(* PLC project TON_TEST, Actility iec61131 1.0.26, author Laurent Nicq *)
(* stored: creationDateTime 2013-01-02T13:55:36, version 1.0.0, modificationDateTime 2013-07-30T14:58:25 *)

PROGRAM main
  VAR_EXTERNAL
    SENSOR : BOOL;
    START : BOOL;
  END_VAR
  VAR
    DELAY : TIME := T#10s;
    Counter : TIME;
  END_VAR
  VAR_EXTERNAL
    TimeElapsed : BOOL;
  END_VAR
  VAR
    OnDelay : TON;
  END_VAR

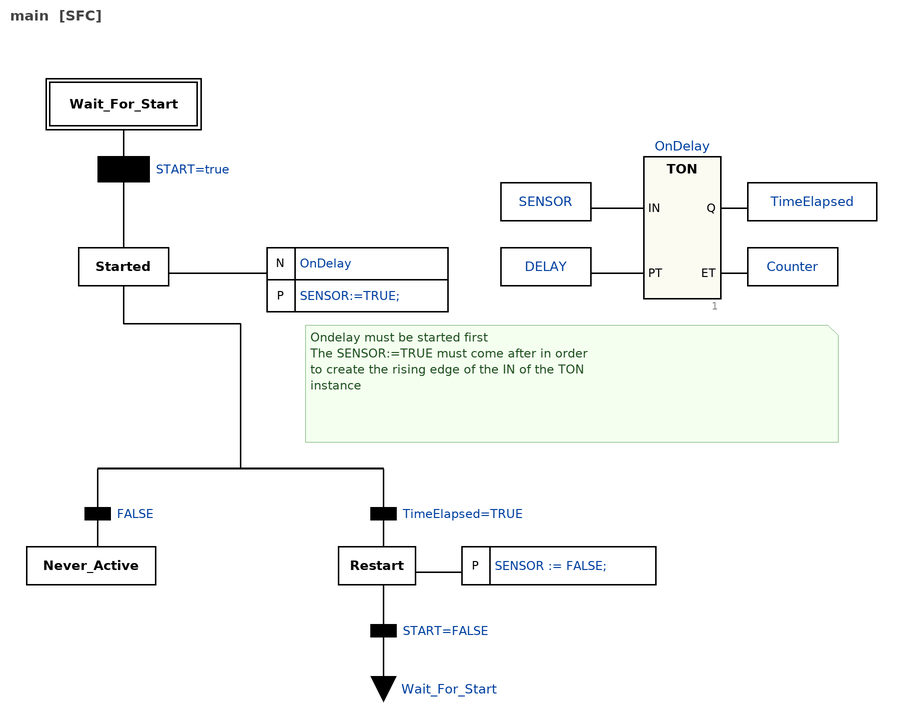
(* Ondelay must be started first
The SENSOR:=TRUE must come after in order
to create the rising edge of the IN of the TON
instance *)
INITIAL_STEP Wait_For_Start:
  COMPUTE_FUNCTION_BLOCKS(S);
END_STEP
TRANSITION FROM Wait_For_Start TO Started
  := START=true;
END_TRANSITION
STEP Started:
  OnDelay(N);
  STARTED_INLINE1(P);
END_STEP
ACTION STARTED_INLINE1:
  SENSOR:=TRUE;
END_ACTION
TRANSITION FROM Started TO Never_Active
  := FALSE;
END_TRANSITION
TRANSITION FROM Started TO Restart
  := TimeElapsed=TRUE;
END_TRANSITION
STEP Never_Active:
END_STEP
STEP Restart:
  RESTART_INLINE2(P);
END_STEP
ACTION RESTART_INLINE2:
  SENSOR := FALSE;
END_ACTION
TRANSITION FROM Restart TO Wait_For_Start
  := START=FALSE;
END_TRANSITION
ACTION COMPUTE_FUNCTION_BLOCKS:  (* blocks drawn on the SFC sheet *)
  OnDelay(IN := SENSOR, PT := DELAY);
  TimeElapsed := OnDelay.Q;
  Counter := OnDelay.ET;
END_ACTION
END_PROGRAM

CONFIGURATION STD_CONF
  VAR_GLOBAL
    SENSOR AT %IXRight : BOOL;
    START AT %IXLeft : BOOL;
    TimeElapsed AT %QXRelay : BOOL;
  END_VAR
  RESOURCE STD_RESSOURCE ON PLC
    TASK STD_TASK(INTERVAL := T#500ms, PRIORITY := 0);
    PROGRAM main WITH STD_TASK : main;
  END_RESOURCE
END_CONFIGURATION
